SUBAPPLICATION Uebung_003 (* Subapplication Type *)
  (* Standard: 61499-2 *)
  (* Version 1.0, 2023-10-23, franz *)
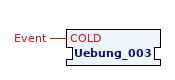
  EVENT_INPUT
    COLD;
  END_EVENT
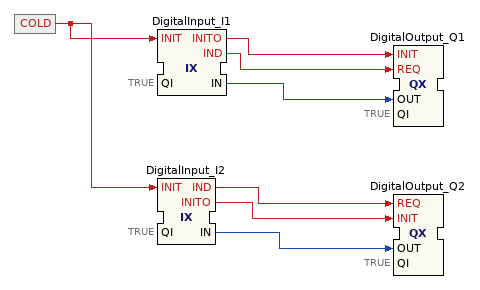
  FBS
    DigitalOutput_Q1 : QX(QI := TRUE);
    DigitalInput_I1 : IX(QI := TRUE);
    DigitalOutput_Q2 : QX(QI := TRUE);
    DigitalInput_I2 : IX(QI := TRUE);
  END_FBS
  EVENT_CONNECTIONS
    COLD TO DigitalInput_I1.INIT;
    DigitalInput_I1.INITO TO DigitalOutput_Q1.INIT;
    DigitalInput_I1.IND TO DigitalOutput_Q1.REQ;
    COLD TO DigitalInput_I2.INIT;
    DigitalInput_I2.IND TO DigitalOutput_Q2.REQ;
    DigitalInput_I2.INITO TO DigitalOutput_Q2.INIT;
  END_CONNECTIONS
  DATA_CONNECTIONS
    DigitalInput_I1.IN TO DigitalOutput_Q1.OUT;
    DigitalInput_I2.IN TO DigitalOutput_Q2.OUT;
  END_CONNECTIONS
END_SUBAPPLICATION
